(* PLC project Progetto_Domotica, Sconosciuto Senza_nome 1 *)
(* stored: creationDateTime 2020-07-06T11:06:18, modificationDateTime 2020-07-16T11:57:43 *)

FUNCTION_BLOCK TP_RESETOFF_TIMER
  VAR_INPUT
    IN : BOOL;
    PT : TIME;
    RESET : BOOL;
  END_VAR
  VAR_OUTPUT
    Q : BOOL;
    ET : TIME := T#0s;
  END_VAR
  VAR
    STATE : SINT := 0;
    PREV_IN : BOOL := FALSE;
    CURRENT_TIME : TIME;
    START_TIME : TIME;
  END_VAR

            (* Pragma to set current time *)
{__SET_VAR(data__->,CURRENT_TIME,,__CURRENT_TIME)}

(*Timer block code *)
IF ((STATE = 0) AND NOT(PREV_IN) AND IN) THEN  (* found rising edge on IN *)
    (* start timer... *)
    STATE := 1;
    Q := TRUE;
    START_TIME := CURRENT_TIME;

ELSIF (STATE = 1) THEN (* timer counting *)
    IF ((START_TIME + PT) <= CURRENT_TIME) THEN (* timer expired *)
        STATE := 2;
        Q := FALSE;
        ET := PT;
    ELSE (* continue counting *)
        ET := CURRENT_TIME - START_TIME;
    END_IF;
END_IF;

IF ((STATE = 2) AND NOT(IN)) THEN
    ET := T#0s;
    STATE := 0;
END_IF;

IF (RESET) THEN (* reset pressed *)
  ET := T#0s;
  STATE := 0;
  Q := FALSE;
END_IF;

PREV_IN := IN;
          
END_FUNCTION_BLOCK

FUNCTION_BLOCK TP_RESET_TIMER
  VAR_INPUT
    IN : BOOL;
    PT : TIME;
    RESET : BOOL;
  END_VAR
  VAR_OUTPUT
    Q : BOOL;
    ET : TIME := T#0s;
  END_VAR
  VAR
    STATE : SINT := 0;
    PREV_IN : BOOL := FALSE;
    CURRENT_TIME : TIME;
    START_TIME : TIME;
  END_VAR

            (* set del tempo corrente *)
{__SET_VAR(data__->,CURRENT_TIME,,__CURRENT_TIME)}

(*Codice timer*)
IF ((STATE = 0) AND NOT(PREV_IN) AND IN) THEN  (* trova rising edge su IN *)
    (* start timer... *)
    STATE := 1;
    Q := TRUE;
    START_TIME := CURRENT_TIME;

ELSIF (STATE = 1) THEN (* inizio conteggio timer *)
    IF ((START_TIME + PT) <= CURRENT_TIME) THEN (* timer esaurito *)
        STATE := 2;
        Q := FALSE;
        ET := PT;
    ELSE (* continuo conteggio *)
        ET := CURRENT_TIME - START_TIME;
    END_IF;
END_IF;

IF ((STATE = 2) AND NOT(IN)) THEN
    ET := T#0s;
    STATE := 0;
END_IF;

IF (RESET) THEN (* reset timer *)
  ET := T#0s;
  STATE := 1;
  Q := TRUE;
  START_TIME := CURRENT_TIME;
END_IF;

PREV_IN := IN;
          
END_FUNCTION_BLOCK

PROGRAM cancello_esterno
  VAR_EXTERNAL
    BUTTON : BOOL;  (* Bottone cancello *)
  END_VAR
  VAR
    LIGHT AT %QX0.2 : BOOL := 0;  (* Luce cancello *)
    MOT_A AT %QX0.3 : BOOL := 0;  (* Motore di apertura cancello *)
  END_VAR
  VAR_EXTERNAL
    MOT_C : BOOL;  (* Motore di chiusura cancello *)
    ALARM1 : BOOL;  (* Allarme cancelli *)
    ALARM2 : BOOL;  (* Allarme garage *)
    ALARM3 : BOOL;  (* Allarme casa *)
    ALARM4 : BOOL;  (* Allarme incendio garage *)
    FOTOC1 : BOOL;  (* Fotocellula cancello *)
    C_CHIUSO : BOOL;  (* Sensore totale chiusura cancello esterno *)
    C_APERTO : BOOL;  (* Sensore totale apertura cancello esterno *)
  END_VAR
  VAR
    BUTTON1 AT %QX0.8 : BOOL := 0;  (* Bottone garage *)
    MOT_A1 AT %QX0.9 : BOOL := 0;  (* Motore di apertura garage *)
  END_VAR
  VAR_EXTERNAL
    MOT_C1 : BOOL;  (* Motore di chiusura garage *)
    FOTOC2 : BOOL;  (* Fotocellula garage *)
    G_CHIUSO : BOOL;  (* Sensore totale chiusura garage *)
  END_VAR
  VAR
    G_APERTO AT %QX0.13 : BOOL := 0;  (* Sensore totale apertura garage *)
  END_VAR
  VAR_EXTERNAL
    S_MOV1 : BOOL;  (* Sensore di movimento garage *)
  END_VAR
  VAR
    BUTTON2 AT %QX0.15 : BOOL := 0;  (* Bottone pedonale *)
  END_VAR
  VAR_EXTERNAL
    C_PEDONALE : BOOL;  (* Sensore stato chiusura cancello pedonale *)
  END_VAR

(* MOTORIZZAZIONE CANCELLO *)
(* AUTOMAZIONE SENSORI APERTURA E CHIUSURA
CANCELLO *)
(* MOTORIZZAZIONE GARAGE *)
(* AUTOMAZIONE SENSORI APERTURA E CHIUSURA GARAGE *)
(* MOTORIZZAZIONE PEDONALE *)
INITIAL_STEP S0:
END_STEP
TRANSITION FROM S0 TO S0B
  := NOT ALARM1 AND BUTTON;
END_TRANSITION
INITIAL_STEP F0:
END_STEP
TRANSITION FROM F0 TO F1
  := NOT ALARM1 AND BUTTON;
END_TRANSITION
INITIAL_STEP S11:
END_STEP
TRANSITION FROM S11 TO S0B0
  := NOT ALARM2 AND (BUTTON1 OR C_APERTO AND NOT G_APERTO);
END_TRANSITION
INITIAL_STEP F6:
END_STEP
TRANSITION FROM F6 TO F7
  := NOT ALARM2 AND BUTTON1;
END_TRANSITION
INITIAL_STEP F12:
END_STEP
TRANSITION FROM F12 TO F13
  := NOT ALARM1 AND BUTTON2;
END_TRANSITION
STEP S0B:
  C_CHIUSO(R);
END_STEP
TRANSITION FROM S0B TO S1
  := F1.X AND (F1.T>=T#20s);
END_TRANSITION
TRANSITION FROM S0B TO S3
  := F2.X;
END_TRANSITION
STEP F1:
  MOT_A(S);
  BUTTON(R);
  LIGHT(S);
END_STEP
TRANSITION FROM F1 TO F2
  := C_APERTO OR BUTTON;
END_TRANSITION
STEP S1:
  C_APERTO(S);
END_STEP
TRANSITION FROM S1 TO S2
  := F3.X;
END_TRANSITION
STEP S3:
  C_APERTO(R);
END_STEP
TRANSITION FROM S3 TO S4
  := F1.T<=F3.T AND F3.X;
END_TRANSITION
STEP F2:
  MOT_A(R);
  BUTTON(R);
  LIGHT(R);
END_STEP
TRANSITION FROM F2 TO F3
  := BUTTON OR (F2.T>=T#5s);
END_TRANSITION
STEP F3:
  MOT_C(S);
  BUTTON(R);
  LIGHT(S);
END_STEP
TRANSITION FROM F3 TO F4
  := BUTTON OR FOTOC1;
END_TRANSITION
TRANSITION FROM F3 TO F5
  := C_CHIUSO;
END_TRANSITION
STEP S2:
  C_APERTO(R);
END_STEP
TRANSITION FROM S2 TO S4
  := F3.T>=T#20s;
END_TRANSITION
TRANSITION FROM S2 TO S5
  := F4.X;
END_TRANSITION
STEP S5:
END_STEP
TRANSITION FROM S5 TO S1
  := F1.X AND (F1.T>=F3.T);
END_TRANSITION
STEP F4:
  MOT_C(R);
  BUTTON(R);
  LIGHT(R);
END_STEP
TRANSITION FROM F4 TO F1
  := (F2.T>=T#5s) OR BUTTON;
END_TRANSITION
STEP F5:
  MOT_C(R);
  LIGHT(R);
END_STEP
TRANSITION FROM F5 TO F0
  := TRUE;
END_TRANSITION
STEP S4:
  C_CHIUSO(S);
END_STEP
TRANSITION FROM S4 TO S0
  := TRUE;
END_TRANSITION
STEP S0B0:
  G_CHIUSO(R);
END_STEP
TRANSITION FROM S0B0 TO S6
  := F7.X AND (F7.T>=T#15s);
END_TRANSITION
TRANSITION FROM S0B0 TO S8
  := F8.X;
END_TRANSITION
STEP F7:
  MOT_A1(S);
  BUTTON1(R);
END_STEP
TRANSITION FROM F7 TO F8
  := G_APERTO;
END_TRANSITION
STEP F8:
  MOT_A1(R);
END_STEP
TRANSITION FROM F8 TO F9
  := BUTTON1 OR (F8.T>=T#15s) AND NOT S_MOV1;
END_TRANSITION
STEP S6:
  G_APERTO(S);
END_STEP
TRANSITION FROM S6 TO S7
  := F9.X;
END_TRANSITION
STEP S8:
  G_APERTO(R);
END_STEP
TRANSITION FROM S8 TO S9
  := F7.T<=F9.T AND F9.X;
END_TRANSITION
STEP F9:
  MOT_C1(S);
  BUTTON1(R);
END_STEP
TRANSITION FROM F9 TO F10
  := BUTTON1 OR FOTOC2;
END_TRANSITION
TRANSITION FROM F9 TO F11
  := G_CHIUSO;
END_TRANSITION
STEP S7:
  G_APERTO(R);
END_STEP
TRANSITION FROM S7 TO S9
  := F9.T>=T#15s;
END_TRANSITION
TRANSITION FROM S7 TO S10
  := F10.X;
END_TRANSITION
STEP S10:
END_STEP
TRANSITION FROM S10 TO S6
  := F7.X AND (F7.T>=F9.T);
END_TRANSITION
STEP F10:
  MOT_C1(R);
  BUTTON1(R);
END_STEP
TRANSITION FROM F10 TO F7
  := (F8.T>=T#5s) OR BUTTON1;
END_TRANSITION
STEP F11:
  MOT_C1(R);
END_STEP
TRANSITION FROM F11 TO F6
  := TRUE;
END_TRANSITION
STEP S9:
  G_CHIUSO(S);
END_STEP
TRANSITION FROM S9 TO S11
  := TRUE;
END_TRANSITION
STEP F13:
  C_PEDONALE(SL, T#10s);
  BUTTON2(R);
END_STEP
TRANSITION FROM F13 TO F12
  := TRUE;
END_TRANSITION
END_PROGRAM

PROGRAM illuminazione
  VAR_EXTERNAL
    C_CHIUSO : BOOL;  (* Sensore totale chiusura cancello esterno *)
    BUTTON : BOOL;  (* Bottone cancello esterno *)
    C_PEDONALE : BOOL;  (* Sensore stato chiusura cancello pedonale *)
    G_CHIUSO : BOOL;  (* Sensore totale chiusura garage *)
    LIGHT1 : BOOL;  (* Luci percorso carrabile *)
    LIGHT2 : BOOL;  (* Luci garage *)
    LIGHT3 : BOOL;  (* Luci percorso pedonale *)
    LIGHT4 : BOOL;  (* Luci portico *)
  END_VAR
  VAR
    S_CREPUSCOLARE AT %QX0.21 : BOOL := 0;  (* Sensore crepuscolare *)
    B_LIGHT1 AT %QX0.22 : BOOL := 0;  (* Bottone luci carrabile *)
    B_LIGHT2 AT %QX0.23 : BOOL := 0;  (* Bottone luci garage *)
    B_LIGHT3 AT %QX0.24 : BOOL := 0;  (* Bottone luci pedonale *)
    B_LIGHT4 AT %QX0.25 : BOOL := 0;  (* Bottone luci portico *)
    B_TIMER AT %QX0.26 : BOOL := 0;  (* Bottone accensione/spegnimento timer *)
  END_VAR
  VAR
    TP0 : TP;  (* Timer *)
    TEMPO_ACCENSIONE : TOD := TOD#12:30:00;  (* Ora di accensione timer *)
    DATA_INIZIALE : DT := DT#2020-07-11-12:29:45;  (* Data di inizio simulazione *)
    TEMPO_CORRENTE : TOD;  (* Ora di simulazione *)
    RTC0 : RTC;  (* Clock di simulazione *)
  END_VAR
  VAR_EXTERNAL
    S_MOV1 : BOOL;  (* Sensore di movimento garage *)
  END_VAR
  VAR
    TP_WITH_RESET0 : TP_RESET_TIMER;  (* Timer con estensione temporale in reset *)
    TP_RESETOFF_TIMER0 : TP_RESETOFF_TIMER;  (* Timer luci percorso pedonale con spegnimento in reset *)
    TP_RESETOFF_TIMER1 : TP_RESETOFF_TIMER;  (* Timer luci portico con spegnimento in reset *)
    TP1 : TP;  (* Timer *)
  END_VAR
  VAR
    GIORNODOPO AT %QX0.50 : BOOL := 0;  (* Ai fini della simulazione per far resettare le variabili temporali *)
  END_VAR

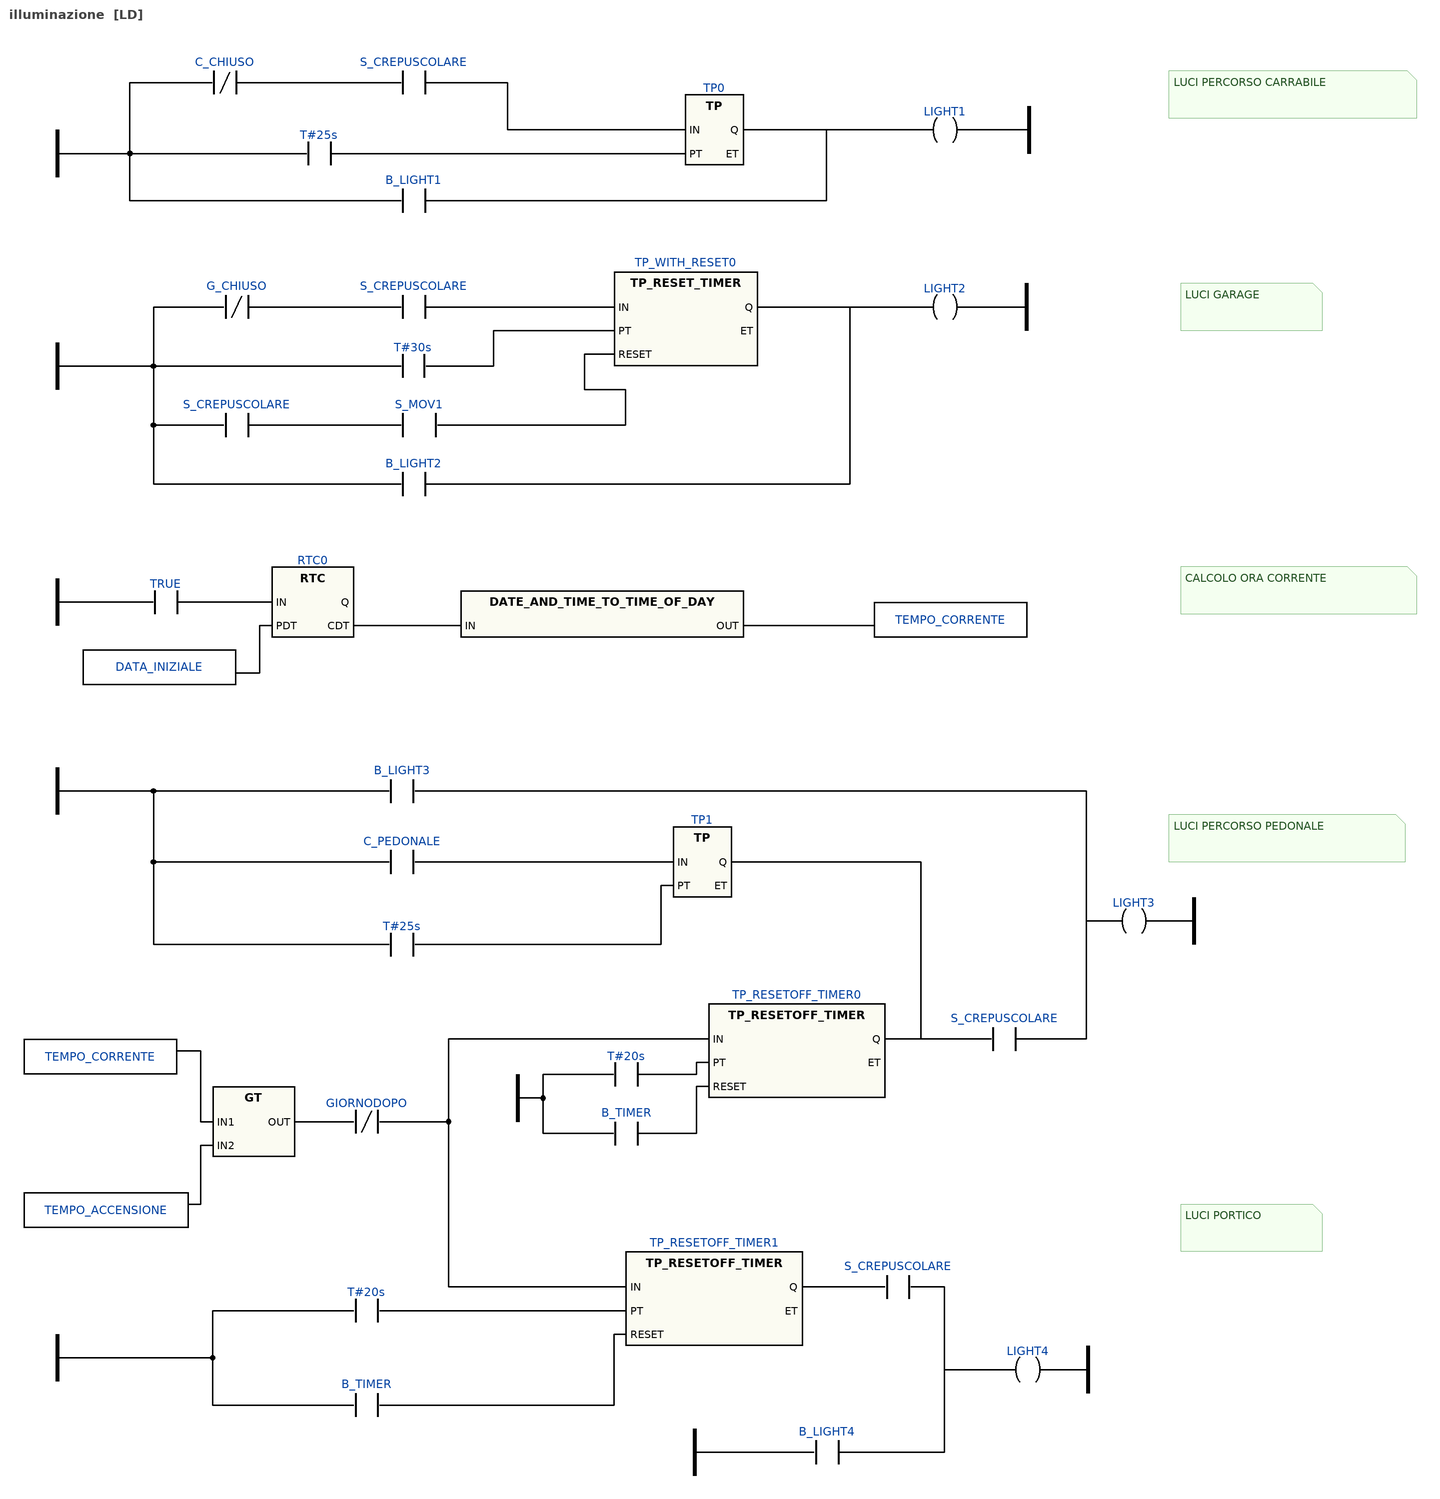
(* LD diagram, written out as Structured Text *)
(* LUCI PERCORSO CARRABILE *)
TP0(IN := NOT C_CHIUSO AND S_CREPUSCOLARE, PT := T#25s);
LIGHT1 := TP0.Q OR B_LIGHT1;
(* LUCI GARAGE *)
TP_WITH_RESET0(IN := NOT G_CHIUSO AND S_CREPUSCOLARE, PT := T#30s, RESET := S_CREPUSCOLARE AND S_MOV1);
LIGHT2 := TP_WITH_RESET0.Q OR B_LIGHT2;
(* CALCOLO ORA CORRENTE *)
RTC0(IN := TRUE, PDT := DATA_INIZIALE);
TEMPO_CORRENTE := DATE_AND_TIME_TO_TIME_OF_DAY(RTC0.CDT);
(* LUCI PERCORSO PEDONALE *)
TP_RESETOFF_TIMER0(IN := TEMPO_CORRENTE > TEMPO_ACCENSIONE AND NOT GIORNODOPO, PT := T#20s, RESET := B_TIMER);
TP1(IN := C_PEDONALE, PT := T#25s);
LIGHT3 := B_LIGHT3 OR (TP_RESETOFF_TIMER0.Q OR TP1.Q) AND S_CREPUSCOLARE;
(* LUCI PORTICO *)
TP_RESETOFF_TIMER1(IN := TEMPO_CORRENTE > TEMPO_ACCENSIONE AND NOT GIORNODOPO, PT := T#20s, RESET := B_TIMER);
LIGHT4 := B_LIGHT4 OR TP_RESETOFF_TIMER1.Q AND S_CREPUSCOLARE;
END_PROGRAM

PROGRAM antifurto
  VAR
    ANTI_THEFT1 AT %QX0.27 : BOOL := 0;  (* Sicurezza cancello esterno *)
    ANTI_THEFT2 AT %QX0.28 : BOOL := 0;  (* Sicurezza garage *)
    ANTI_THEFT3 AT %QX0.29 : BOOL := 0;  (* Sicurezza casa *)
    ANTI_THEFT4 AT %QX0.30 : BOOL := 0;  (* Sicurezza totale *)
    T_PROX1 AT %QX0.31 : BOOL := 0;  (* Telecamera rilevazione prossimità nei pressi del cancello *)
  END_VAR
  VAR_EXTERNAL
    FOTOC1 : BOOL;  (* Fotocellula cancello *)
    FOTOC2 : BOOL;  (* Fotocellula garage *)
    S_MOV1 : BOOL;  (* Sensore movimento garage *)
  END_VAR
  VAR
    S_MOV2 AT %QX0.32 : BOOL := 0;  (* Sensore movimento portico *)
    S_FUMO AT %QX0.33 : BOOL := 0;  (* Rilevatore di fumo garage *)
  END_VAR
  VAR_EXTERNAL
    ALARM1 : BOOL;  (* Allarme cancellI *)
    ALARM2 : BOOL;  (* Allarme garage *)
    ALARM3 : BOOL;  (* Allarme casa *)
    ALARM4 : BOOL;  (* Allarme incendio garage *)
  END_VAR
  VAR
    L_PORTA AT %QX0.38 : BOOL := 0;  (* Serratura elettrica porta *)
    L_FINESTRE AT %QX0.39 : BOOL := 0;  (* Serranda finestre *)
  END_VAR
  VAR_EXTERNAL
    C_CHIUSO : BOOL;  (* Sensore totale chiusura cancello esterno *)
    G_CHIUSO : BOOL;  (* Sensore totale chiusura garage *)
    C_PEDONALE : BOOL;  (* Serratura elettrica pedonale *)
  END_VAR
  VAR
    FARO1 AT %QX0.43 : BOOL := 0;  (* Luci carrabile *)
    FARO2 AT %QX0.44 : BOOL := 0;  (* Luci garage *)
    FARO3 AT %QX0.45 : BOOL := 0;  (* Luci pedonale *)
    FARO4 AT %QX0.46 : BOOL := 0;  (* Luci portico *)
    LIGHT5 AT %QX0.40 : BOOL := 0;  (* Luce fumo garage *)
    SPEAKER1 AT %QX0.41 : BOOL := 0;  (* Speaker allarme *)
    SPRINKLER AT %QX0.42 : BOOL := 0;  (* Sprinkler garage *)
  END_VAR
  VAR
    TON0 : TON;
    TOF0 : TOF;
    TON1 : TON;
    TOF1 : TOF;
    TON2 : TON;
    TOF2 : TOF;
    TON3 : TON;
    TOF3 : TOF;
    TON4 : TON;
    TOF4 : TOF;
  END_VAR

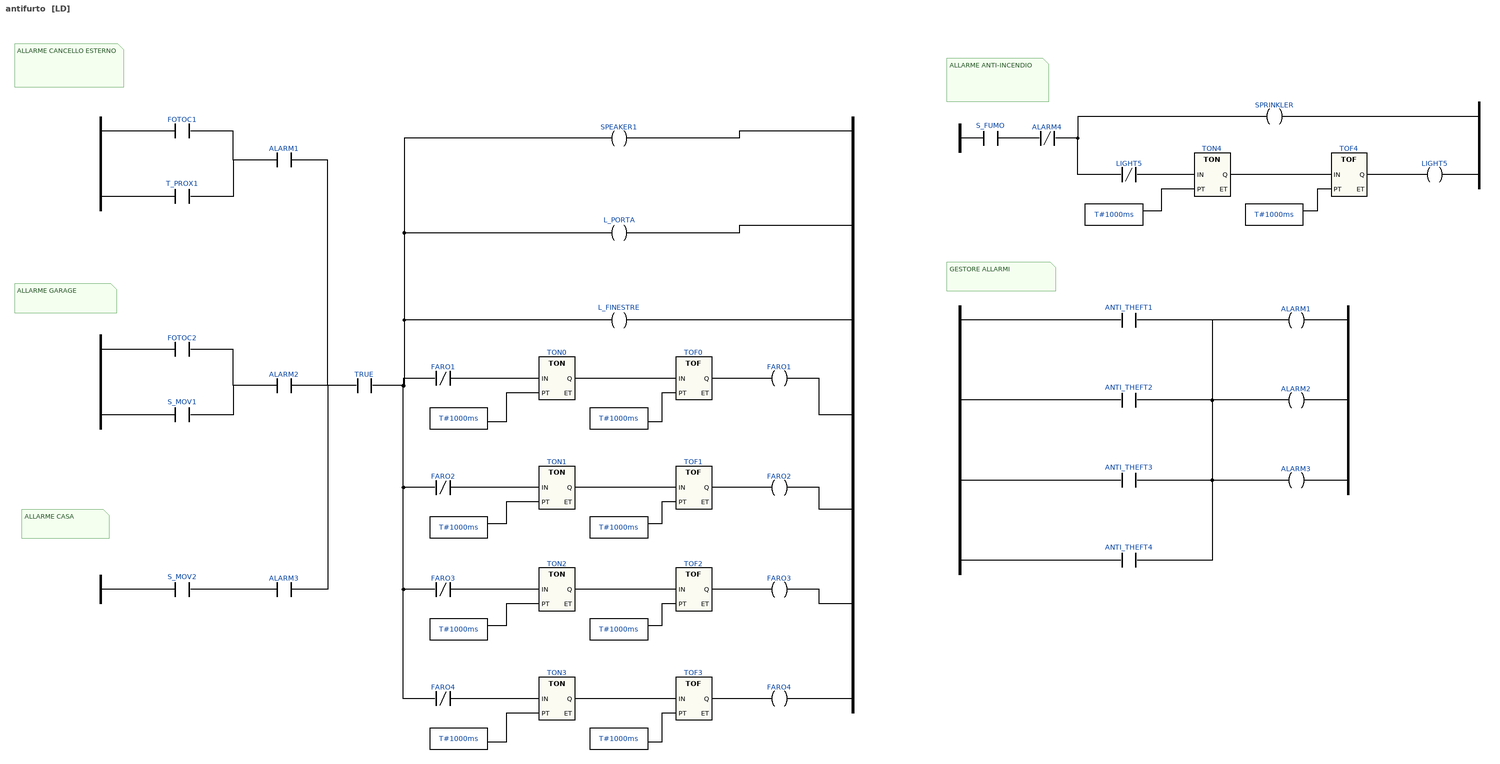
(* LD diagram, written out as Structured Text *)
(* ALLARME CANCELLO ESTERNO *)
(* ALLARME ANTI-INCENDIO *)
SPRINKLER := S_FUMO AND NOT ALARM4;
SPEAKER1 := ((T_PROX1 OR FOTOC1) AND ALARM1 OR (S_MOV1 OR FOTOC2) AND ALARM2 OR S_MOV2 AND ALARM3) AND TRUE;
TON4(IN := S_FUMO AND NOT ALARM4 AND NOT LIGHT5, PT := T#1000ms);
TOF4(IN := TON4.Q, PT := T#1000ms);
LIGHT5 := TOF4.Q;
L_PORTA := ((T_PROX1 OR FOTOC1) AND ALARM1 OR (S_MOV1 OR FOTOC2) AND ALARM2 OR S_MOV2 AND ALARM3) AND TRUE;
(* GESTORE ALLARMI *)
(* ALLARME GARAGE *)
L_FINESTRE := ((T_PROX1 OR FOTOC1) AND ALARM1 OR (S_MOV1 OR FOTOC2) AND ALARM2 OR S_MOV2 AND ALARM3) AND TRUE;
ALARM1 := ANTI_THEFT1 OR ANTI_THEFT4;
TON0(IN := ((T_PROX1 OR FOTOC1) AND ALARM1 OR (S_MOV1 OR FOTOC2) AND ALARM2 OR S_MOV2 AND ALARM3) AND TRUE AND NOT FARO1, PT := T#1000ms);
TOF0(IN := TON0.Q, PT := T#1000ms);
FARO1 := TOF0.Q;
ALARM2 := ANTI_THEFT2 OR ANTI_THEFT4;
ALARM3 := ANTI_THEFT3 OR ANTI_THEFT4;
TON1(IN := ((T_PROX1 OR FOTOC1) AND ALARM1 OR (S_MOV1 OR FOTOC2) AND ALARM2 OR S_MOV2 AND ALARM3) AND TRUE AND NOT FARO2, PT := T#1000ms);
TOF1(IN := TON1.Q, PT := T#1000ms);
FARO2 := TOF1.Q;
(* ALLARME CASA *)
TON2(IN := ((T_PROX1 OR FOTOC1) AND ALARM1 OR (S_MOV1 OR FOTOC2) AND ALARM2 OR S_MOV2 AND ALARM3) AND TRUE AND NOT FARO3, PT := T#1000ms);
TOF2(IN := TON2.Q, PT := T#1000ms);
FARO3 := TOF2.Q;
TON3(IN := ((T_PROX1 OR FOTOC1) AND ALARM1 OR (S_MOV1 OR FOTOC2) AND ALARM2 OR S_MOV2 AND ALARM3) AND TRUE AND NOT FARO4, PT := T#1000ms);
TOF3(IN := TON3.Q, PT := T#1000ms);
FARO4 := TOF3.Q;
END_PROGRAM

CONFIGURATION Config0
  VAR_GLOBAL
    BUTTON AT %QX0.1 : BOOL := 0;
    ALARM1 AT %QX0.34 : BOOL := 0;
    ALARM2 AT %QX0.35 : BOOL := 0;
    ALARM3 AT %QX0.36 : BOOL := 0;
    ALARM4 AT %QX0.37 : BOOL := 0;
    FOTOC1 AT %QX0.5 : BOOL := 0;
    FOTOC2 AT %QX0.11 : BOOL := 0;
    S_MOV1 AT %QX0.14 : BOOL := 0;
    MOT_C AT %QX0.4 : BOOL := 0;
    MOT_C1 AT %QX0.10 : BOOL := 0;
    C_APERTO AT %QX0.7 : BOOL := 0;
    C_CHIUSO AT %QX0.6 : BOOL := 1;
    C_PEDONALE AT %QX0.16 : BOOL := 0;
    LIGHT1 AT %QX0.17 : BOOL := 0;
    LIGHT2 AT %QX0.18 : BOOL := 0;
    LIGHT3 AT %QX0.19 : BOOL := 0;
    LIGHT4 AT %QX0.20 : BOOL := 0;
    G_CHIUSO AT %QX0.12 : BOOL := 1;
  END_VAR
  RESOURCE Res0 ON PLC
    TASK task0(INTERVAL := T#20ms, PRIORITY := 0);
    PROGRAM instance0 WITH task0 : cancello_esterno;
    PROGRAM instance1 WITH task0 : illuminazione;
    PROGRAM instance2 WITH task0 : antifurto;
  END_RESOURCE
END_CONFIGURATION
